// TIA Portal project "ACTEA_Ex5_ap" (V15.1)

(* hardware
DEVICE "S7-1200 station_1"  S7-1200 Station
   slot 0: "Rack_0"  S7-1200 Rack  Rack  V1.0
   slot 1: "PLC_1"  CPU 1215C DC/DC/Rly  6ES7 215-1HG31-0XB0  V3.0
   slot 3: "AQ 1x12BIT_1"  AQ1 signal board  6ES7 232-4HA30-0XB0  V1.0
*)

// ===== PLC "PLC_1"  CPU 1215C DC/DC/Rly =====

VAR_GLOBAL   // PLC tag table "Default tag table"
   "System_Byte" AT %MB254 : Byte;
   "FirstScan" AT %M254.0 : Bool;
   "DiagStatusUpdate" AT %M254.1 : Bool;
   "AlwaysTRUE" AT %M254.2 : Bool;
   "AlwaysFALSE" AT %M254.3 : Bool;
   "Clock_Byte" AT %MB255 : Byte;
   "Clock_10Hz" AT %M255.0 : Bool;
   "Clock_5Hz" AT %M255.1 : Bool;
   "Clock_2.5Hz" AT %M255.2 : Bool;
   "Clock_2Hz" AT %M255.3 : Bool;
   "Clock_1.25Hz" AT %M255.4 : Bool;
   "Clock_1Hz" AT %M255.5 : Bool;
   "Clock_0.625Hz" AT %M255.6 : Bool;
   "Clock_0.5Hz" AT %M255.7 : Bool;
   "iCC_BtnStop_S1" AT %I0.0 : Bool;   // Stop Button
   "iCC_BtnStart_S3" AT %I0.2 : Bool;   // Start Button
   "iCC_McbMot_QM1" AT %I1.1 : Bool;   // Motor circuit breaker
   "iCC_ConMot_KM1" AT %I1.2 : Bool;   // Feedback signal contactor
   "oCC_LmpStart_H1" AT %Q0.0 : Bool;   // Lamp start
   "oCC_LmpStop_H3" AT %Q0.2 : Bool;   // Lamp stop
   "oCC_ConMot_KM1" AT %Q0.6 : Bool;   // Contactor motor
   "mMotStarted" AT %M0.0 : Bool;   // Motor started
   "iCC_SwiDolDor_S4" AT %I0.4 : Bool;   // Selection switch DOL DOR
END_VAR

FUNCTION "FC_DOL" : Void   // FC1, FBD
{ S7_Optimized_Access := 'TRUE' }
VERSION : 0.1
BEGIN

REGION Network 1: Start-stop circuit "mMotStarted"
   // Start circuit = Start button
   // Stop circuit = Stop button AND Motor circuit breaker
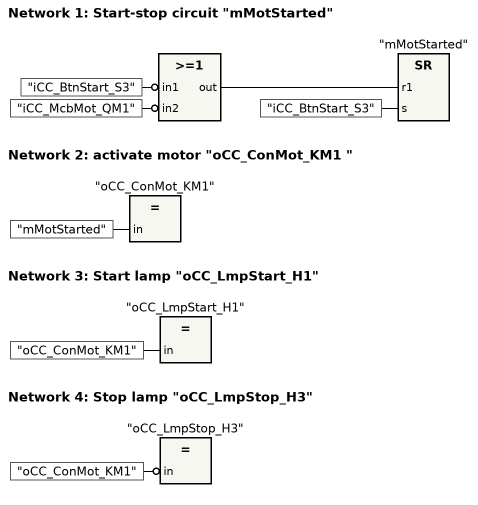
   IF "iCC_BtnStart_S3" THEN
       "mMotStarted" := TRUE;   // SR flip-flop
   END_IF;
   IF NOT "iCC_BtnStart_S3" OR NOT "iCC_McbMot_QM1" THEN "mMotStarted" := FALSE; END_IF;
END_REGION

REGION Network 2: activate motor "oCC_ConMot_KM1 "
   // Motor activation
   "oCC_ConMot_KM1" := "mMotStarted";
END_REGION

REGION Network 3: Start lamp "oCC_LmpStart_H1"
   // contactor feedback signal to (de)activate the green lamp
   "oCC_LmpStart_H1" := "oCC_ConMot_KM1";
END_REGION

REGION Network 4: Stop lamp "oCC_LmpStop_H3"
   // contactor feedback signal to (de)activate the red lamp
   "oCC_LmpStop_H3" := NOT "oCC_ConMot_KM1";
END_REGION
END_FUNCTION

ORGANIZATION_BLOCK "Main"   // OB1, LAD, ProgramCycle
TITLE = "Main Program Sweep (Cycle)"
{ S7_Optimized_Access := 'TRUE' }
VERSION : 0.1
BEGIN

REGION Network 1
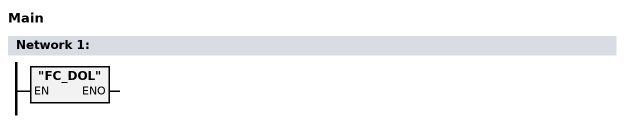
   RUNG wire#powerrail
      "FC_DOL"()
   END_RUNG
   // the same network as SCL:
   "FC_DOL"();
END_REGION
END_ORGANIZATION_BLOCK